PROGRAM MAIN
VAR
	straTestStringArray	: ARRAY [1..10] OF STRING(255);
	fbFillArray	: FB_FillTestArray;
	fbWriteArray	: FB_WriteStringArrayToFile;
	
	bTestFillArray	: BOOL;
	bTestWriteArray	: BOOL;
	
	bTestOpen		: BOOL;
	bTestClose		: BOOL;
	
	fbFileOpen		: FB_FileOpen;
	fbFileClose		: FB_FileClose;
	
END_VAR

IF(_TaskInfo[GETCURTASKINDEXEX()].FirstCycle) THEN
	; // Do Nothing
END_IF


// Run the fill array FB 
fbFillArray(straArrayToFill	:= straTestStringArray);

// Run the file write array
fbWriteArray(straArrayToWrite	:= straTestStringArray);

IF(bTestFillArray) THEN
	fbFillArray.FillArray();
	bTestFillArray	:= FALSE;
END_IF

IF(bTestWriteArray) THEN
	fbWriteArray.WriteArray('C:\TestFile.txt');
	bTestWriteArray	:= FALSE;
END_IF

// Open the file - create it if it doesn't exist already
fbFileOpen(	sNetId 		:= '',
			sPathName 	:= 'C:\TestOpenFile.txt',
			nMode 		:= FOPEN_MODEAPPEND OR FOPEN_MODEPLUS,
			ePath 		:= PATH_GENERIC,
			bExecute 	:= bTestOpen,	
			tTimeout 	:= T#500MS);
			
// Close the file 
fbFileClose(sNetId :='' ,
			hFile := fbFileOpen.hFile,
			bExecute := fbFileOpen.hFile <> 0 AND bTestClose,
			tTimeout := T#500MS);

END_PROGRAM

(* stored: Version 1.1.0.1, ProductVersion 3.1.4024.12
   POU MAIN: Id {43437237-0656-4031-b5f9-3dc60bed1471}, SpecialFunc None *)
